# EPICS StreamDevice protocol: riesling/riesling/device_config/riesling.proto
Terminator = LF;

GetCurr1 {
	out "r";
	in "%f %*f %*f %*f";
}

GetCurr2 {
	in "%*f %f %*f %*f";
}

GetCurr3 {
	in "%*f %*f %f %*f";
}

GetCurr4 {
	in "%*f %*f %*f %f";
}
